{attribute 'qualified_only'}
{attribute 'strict'}
TYPE DeviationMonitorMode :
(
	Diff := 0, Above, Below
);
END_TYPE

(* stored: Version 1.1.0.1, ProductVersion 3.1.4024.6
   DUT DeviationMonitorMode: Id {1157d9f2-440c-4a1a-ba87-7b04fd3851bf} *)
